PROGRAM AxisHorizontal
VAR_INPUT
	Desired_Speed: INT ;
	Desired_Position: UINT ;
	tolerance: UINT;
END_VAR
VAR
	Axis : ST_Axis := (
		uiCounterValue := INPUT.IW_VGR_CounterValueHorizontal,
		bSetCounter := OUTPUT.QX_VGR_SetCounterHorizontal,
		uiSetCounterValue := OUTPUT.QW_VGR_SetCounterValueHorizontal,
		iControl := VGR.QW_VGR_PWM_Horizontal_Control,
		iPWM := VGR.QW_VGR_PWM_Horizontal_M2,
		bJogMinus := VGR.QX_VGR_M2_HorizontalAxisBackward_Q3,
		bJogPlus := VGR.QX_VGR_M2_HorizontalAxisForward_Q4
	);
	Motor_Direction_Horizontal: Motor_direction;
END_VAR

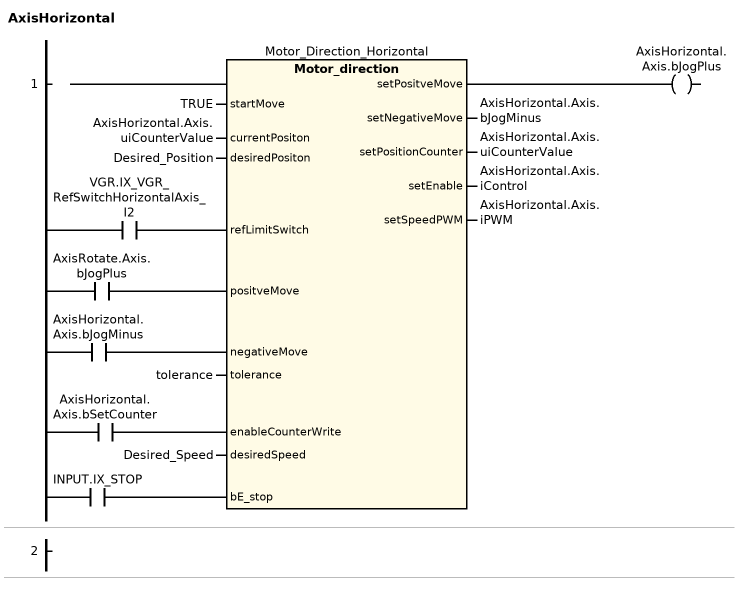
// NETWORK 1
Motor_Direction_Horizontal(
    startMove := TRUE,
    currentPositon := AxisHorizontal.Axis.uiCounterValue,
    desiredPositon := Desired_Position,
    refLimitSwitch := VGR.IX_VGR_RefSwitchHorizontalAxis_I2,
    positveMove := AxisRotate.Axis.bJogPlus,
    negativeMove := AxisHorizontal.Axis.bJogMinus,
    tolerance := tolerance,
    enableCounterWrite := AxisHorizontal.Axis.bSetCounter,
    desiredSpeed := Desired_Speed,
    bE_stop := INPUT.IX_STOP,
    setNegativeMove => AxisHorizontal.Axis.bJogMinus,
    setPositionCounter => AxisHorizontal.Axis.uiCounterValue,
    setEnable => AxisHorizontal.Axis.iControl,
    setSpeedPWM => AxisHorizontal.Axis.iPWM); // Motor_direction
AxisHorizontal.Axis.bJogPlus := Motor_Direction_Horizontal.setPositveMove;

// NETWORK 2

END_PROGRAM

(* stored: Version 1.1.0.1, ProductVersion 3.1.4024.12
   POU AxisHorizontal: Id {7f1b786d-1c4f-41eb-8071-440c25eac7f0}, SpecialFunc None *)
